FUNCTION_BLOCK FB_ST45s
VAR
	_camera : BOOL;
	_sensor	: BOOL;
END_VAR

END_FUNCTION_BLOCK

(* stored: Version 1.1.0.1, ProductVersion 3.1.4024.12
   POU FB_ST45s: Id {a144d5fd-2508-420c-93a0-7793307d38a4}, SpecialFunc None *)
